// TwinCAT 3 PLC project LibPlc
// ProgramVersion: 3.1.4024.0
// libraries:
//   Tc2_Standard, * (Beckhoff Automation GmbH)
//   Tc2_System, * (Beckhoff Automation GmbH)
//   Tc2_TcpIp, * (Beckhoff Automation GmbH)
//   Tc3_Module, * (Beckhoff Automation GmbH)
// project tree:
//   Libraries/Classes/AmeClt/ AmeClt.TcPOU, I_AmeClt.TcIO, P_AmeClt.TcGVL
//   Libraries/Classes/AmeClt/Enums/ E_AssyState.TcDUT (not stored), E_FSM_AmeCltSq.TcDUT, E_FSM_SendRcvSq.TcDUT
//   Libraries/Classes/TcpIp/Client/ E_FSM_TcpIpClt.TcDUT, TcpIpClt.TcPOU
//   Libraries/Functions/ f_StringConcat.TcPOU, f_StringFind.TcPOU, f_StringLeft.TcPOU, f_StringLen.TcPOU, f_StringRight.TcPOU
//   / PlcTask.TcTTO
//   POUs/ APIs.TcPOU, MAIN.TcPOU, Testing.TcPOU
// real-time tasks:
//   TASK PlcTask: cycle T#10ms, priority 20, ADS port 350

CONFIGURATION LibPlc
    RESOURCE PLC ON TwinCAT3
        TASK PlcTask(INTERVAL := T#10ms, PRIORITY := 20);
        PROGRAM MAIN WITH PlcTask : MAIN;
    END_RESOURCE
END_CONFIGURATION

// ---- Libraries/Classes/AmeClt/Enums/E_FSM_AmeCltSq.TcDUT
{attribute 'qualified_only'}
{attribute 'strict'}
TYPE E_FSM_AmeCltSq :
(
	IDLE,
	CREATE_MSG_TO_SEND,
	CALL_SEND_RCV_SQ,
	ERROR,
	DONE
);
END_TYPE

// ---- Libraries/Classes/AmeClt/Enums/E_FSM_SendRcvSq.TcDUT
{attribute 'qualified_only'}
{attribute 'strict'}
TYPE E_FSM_SendRcvSq :
(
	IDLE := 0,
	OPEN_SOCKET,
	SEND_DATA,
	RCV_DATA,
	ERROR,
	DONE
);
END_TYPE

// ---- Libraries/Classes/TcpIp/Client/E_FSM_TcpIpClt.TcDUT
{attribute 'qualified_only'}
{attribute 'strict'}
TYPE E_FSM_TcpIpClt :
(
	IDLE	:= 0,
	OPEN_SOCKET,
	WAIT_SOCKET_OPENED,
	SEND_DATA,
	WAIT_DATA_SENT,
	RECEIVE_DATA,
	WAIT_DATA_RECEIVED,
	CLOSE_SOCKET,
	WAIT_SOCKET_CLOSED,
	ERROR,
	DONE
);
END_TYPE

// ---- Libraries/Classes/AmeClt/P_AmeClt.TcGVL
{attribute 'qualified_only'}
VAR_GLOBAL CONSTANT
	MAX_SIZE_MSG_TO_SEND	:UINT := 1000;
	MAX_SIZE_MSG_TO_RCV		:UINT := 1000;
END_VAR

// ---- Libraries/Classes/AmeClt/I_AmeClt.TcIO
INTERFACE I_AmeClt

METHOD PUBLIC AssyComplete_3011 : BOOL
VAR_INPUT
	sSFC		:STRING;
	eState		:E_AssyState;
	usiOpIndex	:USINT;
END_VAR
END_METHOD

METHOD AssyGetDetails_1026 : BOOL
VAR_INPUT
	sSFC		:STRING;
	usiOpIndex	:USINT;
END_VAR
END_METHOD

PROPERTY sMsgReceived : STRING(P_AmeClt.MAX_SIZE_MSG_TO_RCV)
GET
END_GET
END_PROPERTY

PROPERTY sMsgToSend : STRING(P_AmeClt.MAX_SIZE_MSG_TO_SEND)
GET
END_GET
END_PROPERTY

END_INTERFACE

// ---- POUs/MAIN.TcPOU
PROGRAM MAIN
VAR
	
END_VAR

APIs();
Testing();

END_PROGRAM

// ---- POUs/APIs.TcPOU
PROGRAM APIs
VAR
	_AmeClt	:AmeClt(sSrvNetId := '', sRemoteHost := '192.168.103.17', udiRemotePort := 2001, tTimeout := DEFAULT_ADS_TIMEOUT);
END_VAR

END_PROGRAM

// ---- Libraries/Classes/AmeClt/AmeClt.TcPOU
FUNCTION_BLOCK PUBLIC AmeClt EXTENDS TcpIpClt Implements I_AmeClt
VAR
	_sMsgToSend			:STRING(P_AmeClt.MAX_SIZE_MSG_TO_SEND);
	_sMsgReceived		:STRING(P_AmeClt.MAX_SIZE_MSG_TO_RCV);
	_sSeparator			:STRING(1) 	:= '|';
	_eFSM_SendRcvSqLastState	:E_FSM_SendRcvSq;
	_eFSM_SendRcvSq				:E_FSM_SendRcvSq;
	_eFSM_AmeCltSqLastState		:E_FSM_AmeCltSq;
	_eFSM_AmeCltSq				:E_FSM_AmeCltSq;
END_VAR

VAR CONSTANT
	_sTYPE	:STRING(1) := '1';
END_VAR

METHOD PUBLIC AssyComplete_3011 : BOOL
VAR_INPUT
	sSFC		:STRING;
	eState		:E_AssyState;
	usiOpIndex	:USINT;
END_VAR

VAR
	_sActionCall	:STRING(4) 	:= '3011';
	_sState			:STRING(1);
	_sOpIndex		:STRING(2);
	_bError			:BOOL;
END_VAR
CASE _eFSM_AmeCltSq OF
	E_FSM_AmeCltSq.IDLE:
		IF THIS^._eFSM_SendRcvSq = E_FSM_SendRcvSq.ERROR THEN
			THIS^._eFSM_SendRcvSq := E_FSM_SendRcvSq.IDLE;
		END_IF
		
		THIS^._eFSM_AmeCltSqLastState := E_FSM_AmeCltSq.IDLE;
		THIS^._eFSM_AmeCltSq := E_FSM_AmeCltSq.CREATE_MSG_TO_SEND;
		
	E_FSM_AmeCltSq.CREATE_MSG_TO_SEND:
		_sState	:= INT_TO_STRING(eState);
		_sOpIndex := USINT_TO_STRING(usiOpIndex);
		
		IF NOT _bError AND_THEN NOT f_StringConcat(ADR(THIS^._sTYPE),ADR(THIS^._sSeparator),ADR(THIS^._sMsgToSend),SIZEOF(THIS^._sMsgToSend)) THEN
			_bError := TRUE;
		END_IF
			
		IF NOT _bError AND_THEN NOT f_StringConcat(ADR(THIS^._sMsgToSend),ADR(_sActionCall),ADR(THIS^._sMsgToSend),SIZEOF(THIS^._sMsgToSend)) THEN
			_bError := TRUE;
		END_IF
		
		IF NOT _bError AND_THEN NOT f_StringConcat(ADR(THIS^._sMsgToSend),ADR(THIS^._sSeparator),ADR(THIS^._sMsgToSend),SIZEOF(THIS^._sMsgToSend)) THEN
			_bError := TRUE;
		END_IF
		
		IF NOT _bError AND_THEN NOT f_StringConcat(ADR(THIS^._sMsgToSend),ADR(sSFC),ADR(THIS^._sMsgToSend),SIZEOF(THIS^._sMsgToSend)) THEN
			_bError := TRUE;
		END_IF
		
		IF NOT _bError AND_THEN NOT f_StringConcat(ADR(THIS^._sMsgToSend),ADR(THIS^._sSeparator),ADR(THIS^._sMsgToSend),SIZEOF(THIS^._sMsgToSend)) THEN
			_bError := TRUE;
		END_IF
		
		IF NOT _bError AND_THEN NOT f_StringConcat(ADR(THIS^._sMsgToSend),ADR(_sState),ADR(THIS^._sMsgToSend),SIZEOF(THIS^._sMsgToSend)) THEN
			_bError := TRUE;
		END_IF
		
		IF NOT _bError AND_THEN NOT f_StringConcat(ADR(THIS^._sMsgToSend),ADR(THIS^._sSeparator),ADR(THIS^._sMsgToSend),SIZEOF(THIS^._sMsgToSend)) THEN
			_bError := TRUE;
		END_IF
		
		IF NOT _bError AND_THEN NOT f_StringConcat(ADR(THIS^._sMsgToSend),ADR(_sOpIndex),ADR(THIS^._sMsgToSend),SIZEOF(THIS^._sMsgToSend)) THEN
			_bError := TRUE;
		END_IF
		
		THIS^._eFSM_AmeCltSqLastState := E_FSM_AmeCltSq.CREATE_MSG_TO_SEND;
		THIS^._eFSM_AmeCltSq := E_FSM_AmeCltSq.CALL_SEND_RCV_SQ;
		IF _bError THEN
			THIS^._eFSM_AmeCltSq := E_FSM_AmeCltSq.ERROR;
		END_IF
		
	E_FSM_AmeCltSq.CALL_SEND_RCV_SQ:
		IF SendRcvSq() THEN
			THIS^._eFSM_AmeCltSqLastState := E_FSM_AmeCltSq.CALL_SEND_RCV_SQ;
			THIS^._eFSM_AmeCltSq := E_FSM_AmeCltSq.DONE;
		END_IF
		
		IF bError THEN
			THIS^._eFSM_AmeCltSqLastState := E_FSM_AmeCltSq.CALL_SEND_RCV_SQ;
			THIS^._eFSM_AmeCltSq := E_FSM_AmeCltSq.ERROR;
		END_IF
		
	E_FSM_AmeCltSq.ERROR:
		AssyComplete_3011 := TRUE;
		
	E_FSM_AmeCltSq.DONE:
		AssyComplete_3011 := TRUE;
		
		THIS^._eFSM_AmeCltSqLastState := E_FSM_AmeCltSq.DONE;
		THIS^._eFSM_AmeCltSq := E_FSM_AmeCltSq.IDLE;	
END_CASE
END_METHOD

METHOD PUBLIC AssyGetDetails_1026 : BOOL
VAR_INPUT
	sSFC		:STRING;
	usiOpIndex	:USINT;
END_VAR

VAR
	_sActionCall	:STRING(4) 	:= '1026';
	_sOpIndex		:STRING(2);
	_bError			:BOOL;
END_VAR
CASE _eFSM_AmeCltSq OF
	E_FSM_AmeCltSq.IDLE:
		IF THIS^._eFSM_SendRcvSq = E_FSM_SendRcvSq.ERROR THEN
			THIS^._eFSM_SendRcvSq := E_FSM_SendRcvSq.IDLE;
		END_IF
		
		THIS^._eFSM_AmeCltSqLastState := E_FSM_AmeCltSq.IDLE;
		THIS^._eFSM_AmeCltSq := E_FSM_AmeCltSq.CREATE_MSG_TO_SEND;
		
	E_FSM_AmeCltSq.CREATE_MSG_TO_SEND:
		_sOpIndex := USINT_TO_STRING(usiOpIndex);
		
		IF NOT _bError AND_THEN NOT f_StringConcat(ADR(THIS^._sTYPE),ADR(THIS^._sSeparator),ADR(THIS^._sMsgToSend),SIZEOF(THIS^._sMsgToSend)) THEN
			_bError := TRUE;
		END_IF
			
		IF NOT _bError AND_THEN NOT f_StringConcat(ADR(THIS^._sMsgToSend),ADR(_sActionCall),ADR(THIS^._sMsgToSend),SIZEOF(THIS^._sMsgToSend)) THEN
			_bError := TRUE;
		END_IF
		
		IF NOT _bError AND_THEN NOT f_StringConcat(ADR(THIS^._sMsgToSend),ADR(THIS^._sSeparator),ADR(THIS^._sMsgToSend),SIZEOF(THIS^._sMsgToSend)) THEN
			_bError := TRUE;
		END_IF
		
		IF NOT _bError AND_THEN NOT f_StringConcat(ADR(THIS^._sMsgToSend),ADR(sSFC),ADR(THIS^._sMsgToSend),SIZEOF(THIS^._sMsgToSend)) THEN
			_bError := TRUE;
		END_IF
		
		IF NOT _bError AND_THEN NOT f_StringConcat(ADR(THIS^._sMsgToSend),ADR(THIS^._sSeparator),ADR(THIS^._sMsgToSend),SIZEOF(THIS^._sMsgToSend)) THEN
			_bError := TRUE;
		END_IF
		
		IF NOT _bError AND_THEN NOT f_StringConcat(ADR(THIS^._sMsgToSend),ADR(_sOpIndex),ADR(THIS^._sMsgToSend),SIZEOF(THIS^._sMsgToSend)) THEN
			_bError := TRUE;
		END_IF
		
		THIS^._eFSM_AmeCltSqLastState := E_FSM_AmeCltSq.CREATE_MSG_TO_SEND;
		THIS^._eFSM_AmeCltSq := E_FSM_AmeCltSq.CALL_SEND_RCV_SQ;
		IF _bError THEN
			THIS^._eFSM_AmeCltSq := E_FSM_AmeCltSq.ERROR;
		END_IF
		
	E_FSM_AmeCltSq.CALL_SEND_RCV_SQ:
		IF SendRcvSq() THEN
			THIS^._eFSM_AmeCltSqLastState := E_FSM_AmeCltSq.CALL_SEND_RCV_SQ;
			THIS^._eFSM_AmeCltSq := E_FSM_AmeCltSq.DONE;
		END_IF
		
		IF bError THEN
			THIS^._eFSM_AmeCltSqLastState := E_FSM_AmeCltSq.CALL_SEND_RCV_SQ;
			THIS^._eFSM_AmeCltSq := E_FSM_AmeCltSq.ERROR;
		END_IF
		
	E_FSM_AmeCltSq.ERROR:
		AssyGetDetails_1026 := TRUE;
		
	E_FSM_AmeCltSq.DONE:
		AssyGetDetails_1026 := TRUE;
		
		THIS^._eFSM_AmeCltSqLastState := E_FSM_AmeCltSq.DONE;
		THIS^._eFSM_AmeCltSq := E_FSM_AmeCltSq.IDLE;	
END_CASE
END_METHOD

METHOD PROTECTED SendRcvSq : BOOL
CASE THIS^._eFSM_SendRcvSq OF
	E_FSM_SendRcvSq.IDLE:
		//IF SUPER^._eFSM_TcpIpClt = E_FSM_TcpIpClt.ERROR THEN
		//	SUPER^._eFSM_TcpIpClt := E_FSM_TcpIpClt.IDLE;
		//END_IF
		//
		//THIS^._eFSM_SendRcvSqLastState := E_FSM_SendRcvSq.IDLE;	
		//THIS^._eFSM_SendRcvSq := E_FSM_SendRcvSq.OPEN_SOCKET;
		IF Reset() THEN
			THIS^._eFSM_SendRcvSqLastState := E_FSM_SendRcvSq.IDLE;	
			THIS^._eFSM_SendRcvSq := E_FSM_SendRcvSq.OPEN_SOCKET;
		END_IF
		
	E_FSM_SendRcvSq.OPEN_SOCKET:
		IF OpenSocket() THEN
			THIS^._eFSM_SendRcvSqLastState := E_FSM_SendRcvSq.OPEN_SOCKET;
			THIS^._eFSM_SendRcvSq := E_FSM_SendRcvSq.SEND_DATA;
		END_IF
		
		IF bError THEN
			THIS^._eFSM_SendRcvSqLastState := E_FSM_SendRcvSq.OPEN_SOCKET;
			THIS^._eFSM_SendRcvSq := E_FSM_SendRcvSq.ERROR;
		END_IF
		
	E_FSM_SendRcvSq.SEND_DATA:
		IF Send(ADR(_sMsgToSend), f_StringLen(ADR(_sMsgToSend), SIZEOF(_sMsgToSend))) THEN
			THIS^._eFSM_SendRcvSqLastState := E_FSM_SendRcvSq.SEND_DATA;
			THIS^._eFSM_SendRcvSq := E_FSM_SendRcvSq.RCV_DATA;
		END_IF
		
		IF bError THEN
			THIS^._eFSM_SendRcvSqLastState := E_FSM_SendRcvSq.SEND_DATA;
			THIS^._eFSM_SendRcvSq := E_FSM_SendRcvSq.ERROR;
		END_IF
		
	E_FSM_SendRcvSq.RCV_DATA:
		IF Rcv(ADR(_sMsgReceived), SIZEOF(_sMsgReceived)) THEN
			THIS^._eFSM_SendRcvSqLastState := E_FSM_SendRcvSq.RCV_DATA;
			THIS^._eFSM_SendRcvSq := E_FSM_SendRcvSq.DONE;
		END_IF
		
		IF bError THEN
			THIS^._eFSM_SendRcvSqLastState := E_FSM_SendRcvSq.RCV_DATA;
			THIS^._eFSM_SendRcvSq := E_FSM_SendRcvSq.ERROR;
		END_IF
		
	E_FSM_SendRcvSq.ERROR:
		// Error handling could be implemented here
		SendRcvSq := TRUE;
		
	E_FSM_SendRcvSq.DONE:
		SendRcvSq := TRUE;
		
		THIS^._eFSM_SendRcvSqLastState := E_FSM_SendRcvSq.DONE;
		THIS^._eFSM_SendRcvSq := E_FSM_SendRcvSq.IDLE;
				
END_CASE
END_METHOD

PROPERTY sMsgReceived : STRING(P_AmeClt.MAX_SIZE_MSG_TO_RCV)
GET
sMsgReceived := this^._sMsgReceived;
END_GET
END_PROPERTY

PROPERTY sMsgToSend : STRING(P_AmeClt.MAX_SIZE_MSG_TO_SEND)
GET
sMsgToSend := THIS^._sMsgToSend;
END_GET
END_PROPERTY

END_FUNCTION_BLOCK

// ---- Libraries/Classes/TcpIp/Client/TcpIpClt.TcPOU
FUNCTION_BLOCK PUBLIC TcpIpClt
VAR_INPUT
END_VAR
VAR_OUTPUT
END_VAR
VAR
	// Connection configuration var
	_sSrvNetId			:T_AmsNetId;
	_sRemoteHost		:T_IPv4Addr;
	_udiRemotePort		:UDINT;
	_tTimeOut			:TIME;
	
	_OpenSocket			:FB_SocketConnect;
	_hSocket			:T_HSOCKET;	
	_CloseSocket		:FB_SocketClose;
	_SendData			:FB_SocketSend;
	_RcvData			:FB_SocketReceive;
	
	_bError				:BOOL;
	_udiErrorId			:UDINT;
	
	_eFSM_TcpIpClLastState	:E_FSM_TcpIpClt;
	_eFSM_TcpIpClt			:E_FSM_TcpIpClt;
END_VAR

PROPERTY PUBLIC bError : BOOL
GET
bError := THIS^._bError;
END_GET
END_PROPERTY

METHOD PROTECTED CloseSocket : BOOL
VAR_INST
	_bExecute	:BOOL;
END_VAR
CASE THIS^._eFSM_TcpIpClt OF
	E_FSM_TcpIpClt.IDLE:
		THIS^._bError := FALSE;
		THIS^._udiErrorId := 0;
		
		THIS^._eFSM_TcpIpClLastState := E_FSM_TcpIpClt.IDLE;
		THIS^._eFSM_TcpIpClt := E_FSM_TcpIpClt.CLOSE_SOCKET;
		
	E_FSM_TcpIpClt.CLOSE_SOCKET:
		_bExecute := TRUE;
		
		IF THIS^._CloseSocket.bBusy THEN
			THIS^._eFSM_TcpIpClLastState := E_FSM_TcpIpClt.CLOSE_SOCKET;
			THIS^._eFSM_TcpIpClt := E_FSM_TcpIpClt.WAIT_SOCKET_CLOSED;
			
		END_IF
	
	E_FSM_TcpIpClt.WAIT_SOCKET_CLOSED:
		_bExecute := FALSE;
		
		IF THIS^._CloseSocket.bError THEN
			THIS^._eFSM_TcpIpClLastState := E_FSM_TcpIpClt.WAIT_SOCKET_CLOSED;
			THIS^._eFSM_TcpIpClt := E_FSM_TcpIpClt.ERROR;
			
		ELSIF NOT THIS^._CloseSocket.bBusy THEN
			THIS^._eFSM_TcpIpClLastState := E_FSM_TcpIpClt.WAIT_SOCKET_CLOSED;
			THIS^._eFSM_TcpIpClt := E_FSM_TcpIpClt.DONE;
			
		END_IF
	
	E_FSM_TcpIpClt.ERROR:
		THIS^._bError := TRUE;
		THIS^._udiErrorId := THIS^._CloseSocket.nErrId;
		
		IF NOT THIS^._CloseSocket.bExecute THEN
			CloseSocket := TRUE;
		END_IF
		
	E_FSM_TcpIpClt.DONE:
		
		IF NOT THIS^._CloseSocket.bExecute THEN
			CloseSocket := TRUE;
			THIS^._eFSM_TcpIpClLastState := E_FSM_TcpIpClt.DONE;
			THIS^._eFSM_TcpIpClt := E_FSM_TcpIpClt.IDLE;
		END_IF
END_CASE

THIS^._CloseSocket(
					sSrvNetId	:= THIS^._sSrvNetId, 
					hSocket		:= THIS^._hSocket, 
					bExecute	:= _bExecute, 
					tTimeout	:= THIS^._tTimeOut);
END_METHOD

METHOD PROTECTED ConnConfigUpd : BOOL
VAR_INPUT
	sSrvNetId		:T_AmsNetId;
	sRemoteHost		:T_IPv4Addr;
	udiRemotePort	:UDINT;
	tTimeOut		:TIME;
END_VAR
THIS^._sSrvNetId 		:= sSrvNetId;
THIS^._sRemoteHost		:= sRemoteHost;
THIS^._udiRemotePort	:= udiRemotePort;
THIS^._tTimeOut			:= tTimeOut;
IF THIS^._tTimeOut = T#0S THEN
	THIS^._tTimeOut := DEFAULT_ADS_TIMEOUT;
END_IF
END_METHOD

METHOD FB_init : BOOL
VAR_INPUT
	bInitRetains 	: BOOL; // if TRUE, the retain variables are initialized (warm start / cold start)
	bInCopyCode 	: BOOL;  // if TRUE, the instance afterwards gets moved into the copy code (online change)
	
	sSrvNetId		:T_AmsNetId;
	sRemoteHost		:T_IPv4Addr;
	udiRemotePort	:UDINT;
	tTimeOut		:TIME;
END_VAR
THIS^._sSrvNetId 		:= sSrvNetId;
THIS^._sRemoteHost		:= sRemoteHost;
THIS^._udiRemotePort	:= udiRemotePort;
THIS^._tTimeOut			:= tTimeOut;
IF THIS^._tTimeOut = T#0S THEN
	THIS^._tTimeOut := DEFAULT_ADS_TIMEOUT;
END_IF
END_METHOD

METHOD PROTECTED OpenSocket : BOOL
VAR_INST
	_bExecute	:BOOL;
END_VAR
CASE THIS^._eFSM_TcpIpClt OF
	E_FSM_TcpIpClt.IDLE:
		THIS^._bError := FALSE;
		THIS^._udiErrorId := 0;
		
		THIS^._eFSM_TcpIpClLastState := E_FSM_TcpIpClt.IDLE;
		THIS^._eFSM_TcpIpClt := E_FSM_TcpIpClt.OPEN_SOCKET;
		
	E_FSM_TcpIpClt.OPEN_SOCKET:
		_bExecute := TRUE;
		
		IF THIS^._OpenSocket.bBusy THEN
			THIS^._eFSM_TcpIpClLastState := E_FSM_TcpIpClt.OPEN_SOCKET;
			THIS^._eFSM_TcpIpClt := E_FSM_TcpIpClt.WAIT_SOCKET_OPENED;
			
		END_IF
	
	E_FSM_TcpIpClt.WAIT_SOCKET_OPENED:
		_bExecute := FALSE;
		
		IF THIS^._OpenSocket.bError THEN
			THIS^._eFSM_TcpIpClLastState := E_FSM_TcpIpClt.WAIT_SOCKET_OPENED;
			THIS^._eFSM_TcpIpClt := E_FSM_TcpIpClt.ERROR;
			
		ELSIF NOT THIS^._OpenSocket.bBusy THEN
			THIS^._eFSM_TcpIpClLastState := E_FSM_TcpIpClt.WAIT_SOCKET_OPENED;
			THIS^._eFSM_TcpIpClt := E_FSM_TcpIpClt.DONE;
			
		END_IF
		
	E_FSM_TcpIpClt.ERROR:
		THIS^._bError := TRUE;
		THIS^._udiErrorId := THIS^._OpenSocket.nErrId;
		
		IF NOT THIS^._OpenSocket.bExecute THEN
			OpenSocket := TRUE;
		END_IF	
		
	E_FSM_TcpIpClt.DONE:
		
		IF NOT THIS^._OpenSocket.bExecute THEN
			OpenSocket := TRUE;
			THIS^._eFSM_TcpIpClLastState := E_FSM_TcpIpClt.DONE;
			THIS^._eFSM_TcpIpClt := E_FSM_TcpIpClt.IDLE;
		END_IF
END_CASE

THIS^._OpenSocket(
					sSrvNetId		:= THIS^._sSrvNetId, 
					sRemoteHost		:= THIS^._sRemoteHost, 
					nRemotePort		:= THIS^._udiRemotePort, 
					bExecute		:= _bExecute, 
					tTimeout 		:= THIS^._tTimeOut, 
					hSocket			=> THIS^._hSocket);
END_METHOD

METHOD PROTECTED Rcv : BOOL
VAR_INPUT
	pData	:POINTER TO BYTE;
	udiMaxLen	:UDINT;
END_VAR

VAR_INST
	_bExecute	:BOOL;
END_VAR
CASE THIS^._eFSM_TcpIpClt OF
	E_FSM_TcpIpClt.IDLE:
		THIS^._bError := FALSE;
		THIS^._udiErrorId := 0;
		
		THIS^._eFSM_TcpIpClLastState := E_FSM_TcpIpClt.IDLE;
		THIS^._eFSM_TcpIpClt := E_FSM_TcpIpClt.RECEIVE_DATA;
		
	E_FSM_TcpIpClt.RECEIVE_DATA:
		_bExecute := TRUE;
		
		IF THIS^._RcvData.bBusy THEN
			THIS^._eFSM_TcpIpClLastState := E_FSM_TcpIpClt.RECEIVE_DATA;
			THIS^._eFSM_TcpIpClt := E_FSM_TcpIpClt.WAIT_DATA_RECEIVED;
		END_IF
		
	E_FSM_TcpIpClt.WAIT_DATA_RECEIVED:
		_bExecute := FALSE;
		
		IF THIS^._RcvData.bError THEN
			THIS^._eFSM_TcpIpClLastState := E_FSM_TcpIpClt.WAIT_DATA_RECEIVED;
			THIS^._eFSM_TcpIpClt := E_FSM_TcpIpClt.ERROR;
			
		ELSIF NOT THIS^._RcvData.bBusy THEN
			THIS^._eFSM_TcpIpClLastState := E_FSM_TcpIpClt.WAIT_DATA_RECEIVED;
			THIS^._eFSM_TcpIpClt := E_FSM_TcpIpClt.DONE;
			
		END_IF
		
	E_FSM_TcpIpClt.ERROR:
		THIS^._bError := TRUE;
		THIS^._udiErrorId := THIS^._RcvData.nErrId;
		
		IF NOT THIS^._RcvData.bExecute THEN
			Rcv := TRUE;
		END_IF
		
	E_FSM_TcpIpClt.DONE:
		
		IF NOT THIS^._RcvData.bExecute THEN
			Rcv := TRUE;
			THIS^._eFSM_TcpIpClLastState := E_FSM_TcpIpClt.DONE;
			THIS^._eFSM_TcpIpClt := E_FSM_TcpIpClt.IDLE;
		END_IF	
END_CASE

THIS^._RcvData(
				sSrvNetId	:= THIS^._sSrvNetId, 
				hSocket		:= THIS^._hSocket, 
				cbLen		:= udiMaxLen, 
				pDest		:= pData, 
				bExecute	:= _bExecute, 
				tTimeout	:= THIS^._tTimeOut);
END_METHOD

METHOD PROTECTED Reset : BOOL
VAR_INPUT
END_VAR
THIS^._bError := FALSE;
THIS^._eFSM_TcpIpClt := E_FSM_TcpIpClt.IDLE;

IF NOT THIS^._bError AND THIS^._eFSM_TcpIpClt = E_FSM_TcpIpClt.IDLE THEN
	Reset := TRUE;
END_IF
END_METHOD

METHOD PROTECTED Send : BOOL
VAR_INPUT
	pData	:POINTER TO BYTE;
	udiLen	:UDINT;
END_VAR

VAR_INST
	_bExecute	:BOOL;
END_VAR
CASE THIS^._eFSM_TcpIpClt OF
	E_FSM_TcpIpClt.IDLE:
		THIS^._bError := FALSE;
		THIS^._udiErrorId := 0;
		
		THIS^._eFSM_TcpIpClLastState := E_FSM_TcpIpClt.IDLE;
		THIS^._eFSM_TcpIpClt := E_FSM_TcpIpClt.SEND_DATA;
		
	E_FSM_TcpIpClt.SEND_DATA:
		_bExecute := TRUE;
		
		IF THIS^._SendData.bBusy THEN
			THIS^._eFSM_TcpIpClLastState := E_FSM_TcpIpClt.SEND_DATA;
			THIS^._eFSM_TcpIpClt := E_FSM_TcpIpClt.WAIT_DATA_SENT;
			
		END_IF
	
	E_FSM_TcpIpClt.WAIT_DATA_SENT:
		_bExecute := FALSE;
		
		IF THIS^._SendData.bError THEN
			THIS^._eFSM_TcpIpClLastState := E_FSM_TcpIpClt.WAIT_DATA_SENT;
			THIS^._eFSM_TcpIpClt := E_FSM_TcpIpClt.ERROR;
			
		ELSIF NOT THIS^._SendData.bBusy THEN
			THIS^._eFSM_TcpIpClLastState := E_FSM_TcpIpClt.WAIT_DATA_SENT;
			THIS^._eFSM_TcpIpClt := E_FSM_TcpIpClt.DONE;
			
		END_IF

	E_FSM_TcpIpClt.ERROR:
		THIS^._bError := TRUE;
		THIS^._udiErrorId := THIS^._SendData.nErrId;
		
		IF NOT THIS^._SendData.bExecute THEN
			Send := TRUE;
		END_IF;
		
	E_FSM_TcpIpClt.DONE:
		
		IF NOT THIS^._SendData.bExecute THEN
			Send := TRUE;
			THIS^._eFSM_TcpIpClLastState := E_FSM_TcpIpClt.DONE;
			THIS^._eFSM_TcpIpClt := E_FSM_TcpIpClt.IDLE;
		END_IF
END_CASE

THIS^._SendData(
				sSrvNetId	:= THIS^._sSrvNetId, 
				hSocket		:= THIS^._hSocket, 
				cbLen		:= udiLen, 
				pSrc		:= pData, 
				bExecute	:= _bExecute, 
				tTimeout	:= THIS^._tTimeOut);
END_METHOD

PROPERTY PUBLIC udiErrorId : UDINT
GET
udiErrorId := THIS^._udiErrorId ;
END_GET
END_PROPERTY

END_FUNCTION_BLOCK

// ---- Libraries/Functions/f_StringConcat.TcPOU
FUNCTION f_StringConcat : BOOL
VAR_INPUT
	pSrc1		:POINTER TO BYTE;
	pSrc2		:POINTER TO BYTE;
	pDst		:POINTER TO BYTE;
	udiDstSize	:UDINT;
END_VAR
VAR
	_byNull		:BYTE := 16#00;
	_pSrc1		:POINTER TO BYTE;
	_pSrc2		:POINTER TO BYTE;
	_pDst		:POINTER TO BYTE;
	_udiDstSize	:UDINT;
	_udiIndex	:UDINT;
	_udiIndexStartCleaning :UDINT;
END_VAR

_pSrc1 	:= pSrc1;
_pSrc2 	:= pSrc2;
_pDst 	:= pDst;
_udiDstSize := udiDstSize - 1;

FOR _udiIndex := 1 TO _udiDstSize DO
	IF _pSrc1^ <> _byNull THEN
		// Concatenate Src1 to Dst
		_pDst^ := _pSrc1^;
		
		_pSrc1 := _pSrc1 + SIZEOF(BYTE);
		_pDst := _pDst + SIZEOF(BYTE);
	ELSE
		FOR _udiIndex := _udiIndex TO _udiDstSize DO
			// Concatenate Src1 to Dst
			IF _pSrc2^ <> _byNull THEN
				_pDst^ := _pSrc2^;
				
				_pSrc2 := _pSrc2 + SIZEOF(BYTE);
				_pDst := _pDst + SIZEOF(BYTE);
			ELSE
				JMP lbl_Complete;
			END_IF
			
			IF _udiIndex = _udiDstSize THEN
				JMP lbl_Complete;
			END_IF
		END_FOR	
	END_IF
	
	IF _udiIndex = _udiDstSize THEN
		JMP lbl_Complete;
	END_IF
END_FOR

lbl_Complete:
FOR _udiIndexStartCleaning := _udiIndex TO _udiDstSize DO
	// Cleaning of Dst
	IF _pDst^ <> _byNull THEN
		_pDst^ := _byNull;
		
		_pDst := _pDst + SIZEOF(BYTE);
	ELSE
		EXIT;
	END_IF
END_FOR	

IF _udiIndex <= _udiDstSize AND _udiIndex > 1 (*AND _pSrc1^ = _byNull AND _pSrc2^ = _byNull*) THEN
	f_StringConcat := TRUE;
END_IF

END_FUNCTION

// ---- Libraries/Functions/f_StringLen.TcPOU
FUNCTION f_StringLen : UDINT
VAR_INPUT
	pSrc		:POINTER TO BYTE;
	udiMaxSize	:UDINT;
END_VAR
VAR
	_byNull		:BYTE := 16#00;
	_udiIndex	:UDINT;
END_VAR

FOR _udiIndex := 0 TO udiMaxSize DO
	IF pSrc^ = _byNull THEN
		EXIT;
	END_IF
	
	pSrc := pSrc + SIZEOF(BYTE);
END_FOR

f_StringLen := _udiIndex;

END_FUNCTION

// ---- POUs/Testing.TcPOU
PROGRAM Testing
VAR
	_I_AmeClt				:I_AmeClt := APIs._AmeClt;
	_sSfc					:STRING := 'Testing_SFC';
	_sMsgToSend				:STRING(P_AmeClt.MAX_SIZE_MSG_TO_SEND);
	_sMsgReceived			:STRING(P_AmeClt.MAX_SIZE_MSG_TO_RCV);
	
	_bAssyGetDetails		:BOOL;
	_bAssyComplete			:BOOL;
	_uiAssyCompleteCycles	:UINT;
	
	_sSrc					:STRING(2000) := '1234Hola';
	_sStrToFind				:STRING(10) := '';
	_udiStrToFindIndexPos	:UDINT;
	_bLeft					:BOOL;
	_udiLeftIndex			:UDINT;
	_sStrleft				:STRING;
	_bRight					:BOOL;
	_udiRightIndex			:UDINT;
	_sStrRight				:STRING(2000);
	
	
	
END_VAR

IF _bAssyGetDetails OR _bAssyComplete THEN
	_uiAssyCompleteCycles := _uiAssyCompleteCycles + 1;
END_IF

IF _bAssyComplete  AND_THEN _I_AmeClt.AssyComplete_3011(_sSfc, E_AssyState.PASS, 1) THEN
	_sMsgToSend := _I_AmeClt.sMsgToSend;
	_sMsgReceived := _I_AmeClt.sMsgReceived;
	_bAssyComplete := FALSE;
END_IF

IF _bAssyGetDetails  AND_THEN _I_AmeClt.AssyGetDetails_1026(_sSfc, 1) THEN
	_sMsgToSend := _I_AmeClt.sMsgToSend;
	_sMsgReceived := _I_AmeClt.sMsgReceived;
	_bAssyGetDetails := FALSE;
END_IF

//_udiStrToFindIndexPos := f_StringFind(ADR(_sSrc), SIZEOF(_sSrc), _sStrToFind);
_udiStrToFindIndexPos := f_StringFind(ADR(_sSrc), SIZEOF(_sSrc), 'Handle_00:') + f_StringLen(ADR('Handle_00:'), SIZEOF('Handle_00:'));

_bRight := f_StringRight(ADR(_sSrc), ADR(_sStrRight), SIZEOF(_sStrRight), _udiStrToFindIndexPos);

_bLeft := f_StringLeft(ADR(_sSrc), ADR(_sStrLeft), SIZEOF(_sStrLeft), _udiLeftIndex);

//_bRight := f_StringRight(ADR(_sSrc), ADR(_sStrRight), SIZEOF(_sStrRight), _udiRightIndex);

END_PROGRAM

// ---- Libraries/Functions/f_StringFind.TcPOU
FUNCTION f_StringFind : UDINT
VAR_INPUT
	pSrc		:POINTER TO BYTE;			// string source
	udiSrcSize	:UDINT;						// string length source
	sStrToFind	:STRING(MAX_STRING_LENGTH);
END_VAR
VAR
	_pSrc				:POINTER TO BYTE;
	_udiSrcStrLen		:UDINT;
	_udiStrToFindLen	:UDINT;
	_pStrExtracted		:POINTER TO BYTE;
	_sStrExtracted		:STRING(MAX_STRING_LENGTH);
	
	_udiStrToFindIndex	:UDINT;
	_udiIndex			:UDINT;
END_VAR

_udiSrcStrLen		:= f_StringLen(pSrc,udiSrcSize);
_udiStrToFindLen	:= f_StringLen(ADR(sStrToFind),SIZEOF(sStrToFind));

// if source string length is less that string to find length is not possible execute the logic
IF _udiSrcStrLen < _udiStrToFindLen OR  _udiSrcStrLen = 0 OR _udiStrToFindLen = 0 THEN
	f_StringFind := 0;
	RETURN;
END_IF

_pSrc := pSrc;
REPEAT
	_udiIndex := _udiIndex + 1;	

	_pStrExtracted := ADR(_sStrExtracted);
	FOR _udiStrToFindIndex := 1 TO _udiStrToFindLen DO
		_pStrExtracted^ := _pSrc^;
		_pStrExtracted 	:= _pStrExtracted + SIZEOF(BYTE);
		_pSrc 			:= _pSrc + SIZEOF(BYTE);
	END_FOR
	
	IF sStrToFind = _sStrExtracted THEN
		f_StringFind := _udiIndex;
		EXIT;
	END_IF
	
	_pSrc := pSrc + (_udiIndex * SIZEOF(BYTE));
UNTIL
	_udiIndex > (_udiSrcStrLen - _udiStrToFindLen)
END_REPEAT

IF _udiIndex > (_udiSrcStrLen - _udiStrToFindLen) THEN	// String to find is not existing
	f_StringFind := 0;
END_IF

memset(_pStrExtracted, 16#00, _udiStrToFindLen);

END_FUNCTION

// ---- Libraries/Functions/f_StringRight.TcPOU
FUNCTION f_StringRight : BOOL
VAR_INPUT
	pSrc		:POINTER TO BYTE;	// Source pointer
	pDst		:POINTER TO BYTE;	// Destination pointer
	udiDstSize	:UDINT;				// Destination size
	udiStartPos	:UDINT;
END_VAR
VAR
	_pSrcStartPos	:POINTER TO BYTE;
	_pDst		:POINTER TO BYTE;
	_udiDstSize	:UDINT;
	_byNull		:BYTE := 16#00;
	_udiIndex	:UDINT;
END_VAR

_pSrcStartPos := pSrc + ((udiStartPos - 1) * SIZEOF(BYTE));
_pDst := pDst;
_udiDstSize := udiDstSize - 1;

// Start position must not be cero
IF udiStartPos = 0 THEN
	_udiIndex := 1;
	JMP lbl_CleanDestination;
END_IF

//Extracting data
FOR _udiIndex := 1 TO udiDstSize DO
	IF _pSrcStartPos^ <> _byNull THEN
		_pDst^ := _pSrcStartPos^;
	ELSE
		EXIT;
	END_IF
	
	_pSrcStartPos := _pSrcStartPos + SIZEOF(BYTE);
	_pDst := _pDst + SIZEOF(BYTE);
END_FOR

// Clean destination data
lbl_CleanDestination:
	FOR _udiIndex := _udiIndex TO _udiDstSize DO
		IF _pDst^ <> _byNull THEN
			_pDst^ := _byNull;
		ELSE
			EXIT;
		END_IF
		
		_pDst := _pDst + SIZEOF(BYTE);
	END_FOR
	
	IF udiStartPos <> 0  AND pDst^ <> _byNull THEN
		f_StringRight := TRUE;
	END_IF

END_FUNCTION

// ---- Libraries/Functions/f_StringLeft.TcPOU
FUNCTION f_StringLeft : BOOL
VAR_INPUT
	pSrc		:POINTER TO BYTE;
	pDst		:POINTER TO BYTE;
	udiDstSize	:UDINT;				// Destination size
	udiLen		:UDINT;				// String length to extract
END_VAR
VAR
	_pSrc		:POINTER TO BYTE;
	_pDst		:POINTER TO BYTE;
	_udiDstSize	:UDINT;				// Destination size
	_byNull		:BYTE := 16#00;
	_udiIndex	:UDINT;
END_VAR

_pSrc := pSrc;
_pDst := pDst;
_udiDstSize := udiDstSize - 1;

// String size to extract must not be greater than destination size
IF udiLen > _udiDstSize THEN
	_udiIndex := 1;
	JMP lbl_CleanDestination;
END_IF

// Extracting data
FOR _udiIndex := 1 TO udiLen DO
	IF _pSrc^ <> _byNull THEN
		_pDst^ := _pSrc^;
	ELSE
		EXIT;
	END_IF
	
	_pSrc := _pSrc + SIZEOF(BYTE);
	_pDst := _pDst + SIZEOF(BYTE);
END_FOR

// Clean destination data
lbl_CleanDestination:
	FOR _udiIndex := _udiIndex TO _udiDstSize DO
		IF _pDst^ <> _byNull THEN
			_pDst^ := _byNull;
		ELSE
			EXIT;
		END_IF
		
		_pDst := _pDst + SIZEOF(BYTE);
	END_FOR
	
	IF udiLen <> 0 AND _udiIndex > udiLen THEN
		f_StringLeft := TRUE;
	END_IF

END_FUNCTION
